// Implicitly generated code : DO NOT EDIT
FUNCTION CheckBounds : DINT
VAR_INPUT
	index, lower, upper: DINT;
END_VAR

{noflow}
IF (index < lower) THEN
	CheckBounds := lower;
	F_Log(E_LogLevel.eFatal, 'Check bounds exception: {index} {lower} {upper}').WithLogger('CheckBounds').WithAnyArg(index).WithAnyArg(lower).WithAnyArg(upper).CreateLog();
ELSIF(index > upper) THEN
	CheckBounds := upper;
	F_Log(E_LogLevel.eFatal, 'Check bounds exception: {index} {lower} {upper}').WithLogger('CheckBounds').WithAnyArg(index).WithAnyArg(lower).WithAnyArg(upper).CreateLog();
ELSE
	CheckBounds := index;
END_IF
{flow}

END_FUNCTION

(* stored: Version 1.1.0.1, ProductVersion 3.1.4024.0
   POU CheckBounds: Id {4aa71e58-8a22-49e2-8b69-c56cbe34a862}, SpecialFunc CheckBounds *)
